GLOBALCONSTANTS ISO_CAN_NODEs (* Global constants *)
  (* Standard: 61499-1 *)
  (* Version 1.0, 2025-10-05, franz *)
  PACKAGE isobus::pgn;
  VAR_GLOBAL CONSTANT
    ISO_CAN_NODE1 : USINT := 0; (* CAN 1 *)
    ISO_CAN_NODE2 : USINT := 1; (* CAN 2 *)
    ISO_CAN_NODE3 : USINT := 2; (* CAN 3 *)
    ISO_CAN_NODE4 : USINT := 3; (* CAN 4 *)
  END_VAR
END_GLOBALCONSTANTS
